// SIMATIC S7-200 project (STEP 7-Micro/WIN), CPU 224 REL 01.11

SYMBOL_TABLE USER1
Start            I0.0
stopp            I0.1
A1               Q0.0
B1               Q0.1
A2               Q0.2
B2               Q0.3
END_SYMBOL_TABLE

ORGANIZATION_BLOCK MAIN:OB1
TITLE=PROGRAM COMMENTS
BEGIN
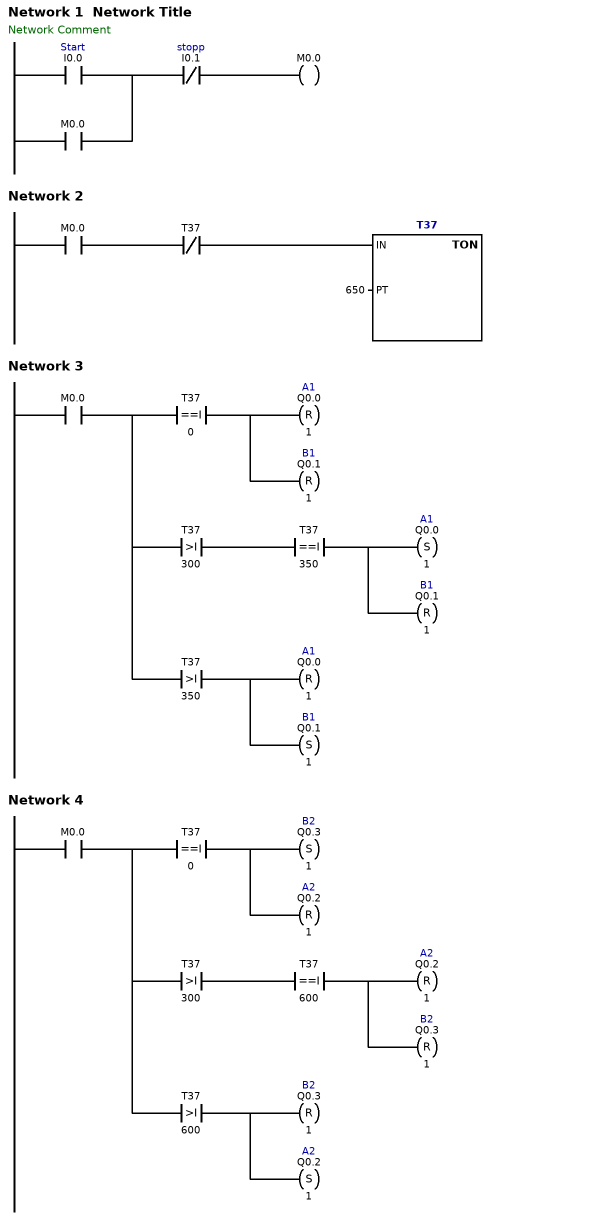
Network 1 // Network Title
// Network Comment
LD     Start:I0.0
O      M0.0
AN     stopp:I0.1
=      M0.0
Network 2
LD     M0.0
AN     T37
TON    T37, 650
Network 3
// (network saved uncompiled; LAD cells follow)
// row 0: c0 -| |- M0.0 v  c1 -|==I|- T37, 0 v  c2 -(R) A1:Q0.0, 1
// row 1: c0 ^v  c1 ^  c2 -(R) B1:Q0.1, 1
// row 2: c0 ^v  c1 -|>I|- T37, 300  c2 -|==I|- T37, 350 v  c3 -(S) A1:Q0.0, 1
// row 3: c0 ^v  c2 ^  c3 -(R) B1:Q0.1, 1
// row 4: c0 ^  c1 -|>I|- T37, 350 v  c2 -(R) A1:Q0.0, 1
// row 5: c1 ^  c2 -(S) B1:Q0.1, 1
Network 4
// (network saved uncompiled; LAD cells follow)
// row 0: c0 -| |- M0.0 v  c1 -|==I|- T37, 0 v  c2 -(S) B2:Q0.3, 1
// row 1: c0 ^v  c1 ^  c2 -(R) A2:Q0.2, 1
// row 2: c0 ^v  c1 -|>I|- T37, 300  c2 -|==I|- T37, 600 v  c3 -(R) A2:Q0.2, 1
// row 3: c0 ^v  c2 ^  c3 -(R) B2:Q0.3, 1
// row 4: c0 ^  c1 -|>I|- T37, 600 v  c2 -(R) B2:Q0.3, 1
// row 5: c1 ^  c2 -(S) A2:Q0.2, 1
END_ORGANIZATION_BLOCK
